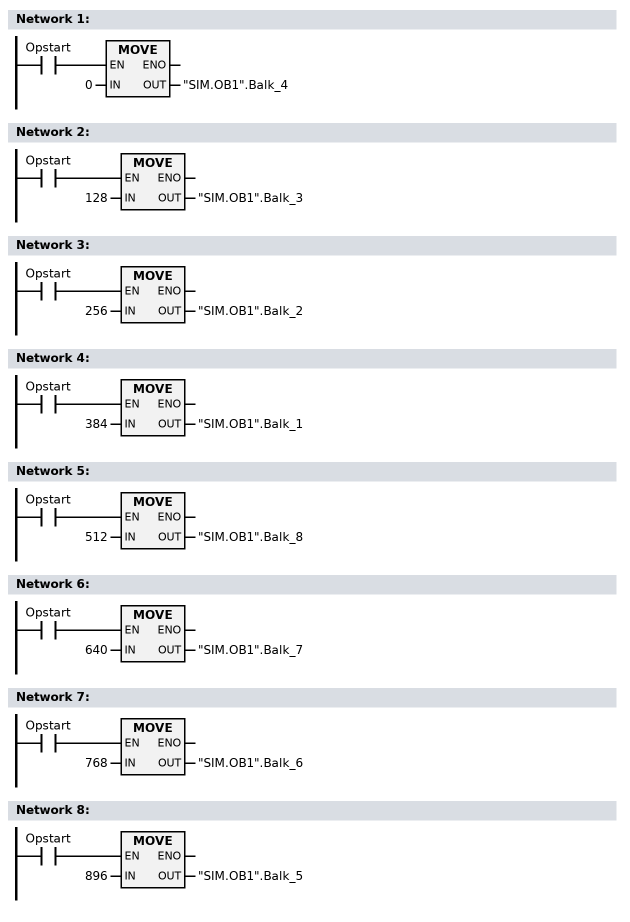
NETWORK
TITLE =
      A     "Opstart";
      JNB   _001;
      L     0;
      T     "SIM.OB1".Balk_4;
_001: NOP   0;
NETWORK
TITLE =
      A     "Opstart";
      JNB   _002;
      L     128;
      T     "SIM.OB1".Balk_3;
_002: NOP   0;
NETWORK
TITLE =
      A     "Opstart";
      JNB   _003;
      L     256;
      T     "SIM.OB1".Balk_2;
_003: NOP   0;
NETWORK
TITLE =
      A     "Opstart";
      JNB   _004;
      L     384;
      T     "SIM.OB1".Balk_1;
_004: NOP   0;
NETWORK
TITLE =
      A     "Opstart";
      JNB   _005;
      L     512;
      T     "SIM.OB1".Balk_8;
_005: NOP   0;
NETWORK
TITLE =
      A     "Opstart";
      JNB   _006;
      L     640;
      T     "SIM.OB1".Balk_7;
_006: NOP   0;
NETWORK
TITLE =
      A     "Opstart";
      JNB   _007;
      L     768;
      T     "SIM.OB1".Balk_6;
_007: NOP   0;
NETWORK
TITLE =
      A     "Opstart";
      JNB   _008;
      L     896;
      T     "SIM.OB1".Balk_5;
_008: NOP   0;
END_FUNCTION

FUNCTION "SIM.user" : VOID	// FC 11
VERSION : 0.1
BEGIN
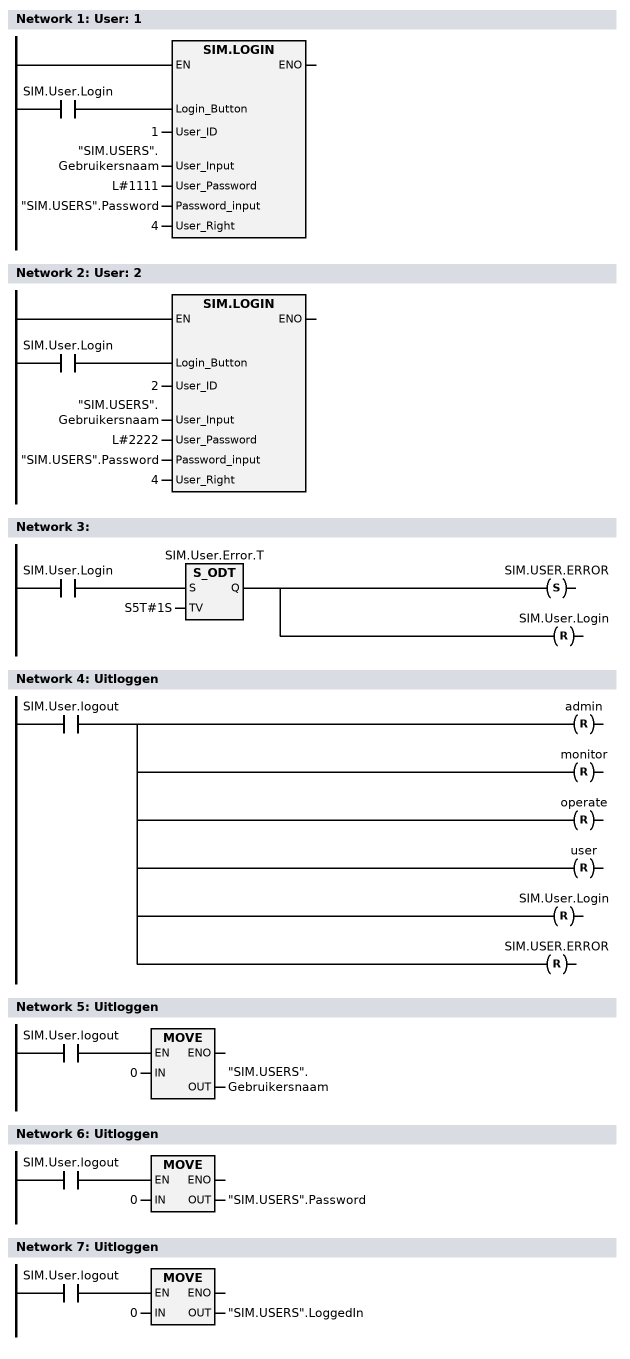
NETWORK
TITLE = User: 1
      A     "SIM.User.Login";
      =     L 0.0;
      BLD   103;
      CALL  "SIM.LOGIN" (
           Login_Button             := L 0.0,
           User_ID                  := 1,
           User_Input               := "SIM.USERS".Gebruikersnaam,
           User_Password            := L#1111,
           Password_input           := "SIM.USERS".Password,
           User_Right               := 4);
      NOP   0;
NETWORK
TITLE = User: 2
      A     "SIM.User.Login";
      =     L 0.0;
      BLD   103;
      CALL  "SIM.LOGIN" (
           Login_Button             := L 0.0,
           User_ID                  := 2,
           User_Input               := "SIM.USERS".Gebruikersnaam,
           User_Password            := L#2222,
           Password_input           := "SIM.USERS".Password,
           User_Right               := 4);
      NOP   0;
NETWORK
TITLE =
      A     "SIM.User.Login";
      L     S5T#1S;
      SD    "SIM.User.Error.T";
      NOP   0;
      NOP   0;
      NOP   0;
      A     "SIM.User.Error.T";
      S     "SIM.USER.ERROR";
      R     "SIM.User.Login";
NETWORK
TITLE = Uitloggen
      A     "SIM.User.logout";
      R     "admin";
      R     "monitor";
      R     "operate";
      R     "user";
      R     "SIM.User.Login";
      R     "SIM.USER.ERROR";
NETWORK
TITLE = Uitloggen
      A     "SIM.User.logout";
      JNB   _001;
      L     0;
      T     "SIM.USERS".Gebruikersnaam;
_001: NOP   0;
NETWORK
TITLE = Uitloggen
      A     "SIM.User.logout";
      JNB   _002;
      L     0;
      T     "SIM.USERS".Password;
_002: NOP   0;
NETWORK
TITLE = Uitloggen
      A     "SIM.User.logout";
      JNB   _003;
      L     0;
      T     "SIM.USERS".LoggedIn;
_003: NOP   0;
END_FUNCTION

FUNCTION "Positionering_balken" : VOID	// FC 12
VERSION : 0.1
BEGIN
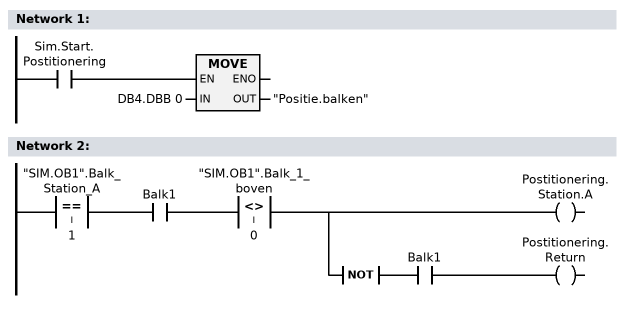
NETWORK
TITLE =
      A     "Sim.Start.Postitionering";
      JNB   _001;
      L     DB4.DBB 0;
      T     "Positie.balken";
_001: NOP   0;
NETWORK
TITLE =
      A(;
      L     "SIM.OB1".Balk_Station_A;
      L     1;
      ==I;
      );
      A     "Balk1";
      A(;
      L     "SIM.OB1".Balk_1_boven;
      L     0;
      <>I;
      );
      =     L 0.0;
      A     L 0.0;
      BLD   102;
      =     "Postitionering.Station.A";
      A     L 0.0;
      NOT;
      A     "Balk1";
      =     "Postitionering.Return";
END_FUNCTION

FUNCTION "Sub_routine" : VOID	// FC 14
VERSION : 0.1
VAR_INPUT
  voorwaarde : BOOL ;
END_VAR
VAR_IN_OUT
  huidige : BOOL ;
  volgende : BOOL ;
END_VAR
BEGIN
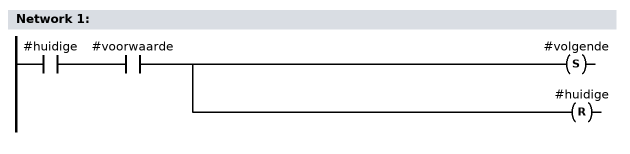
NETWORK
TITLE =
      A     #huidige;
      A     #voorwaarde;
      S     #volgende;
      R     #huidige;
END_FUNCTION

FUNCTION "Opstart_subroutine" : VOID	// FC 15
VERSION : 0.1
VAR_INPUT
  voorwaarde : BOOL ;
END_VAR
VAR_IN_OUT
  huidige : BOOL ;
  volgende_1 : BOOL ;
  volgende_2 : BOOL ;
END_VAR
BEGIN
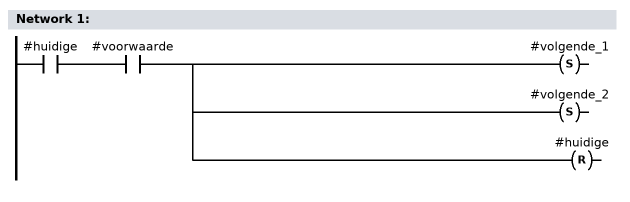
NETWORK
TITLE =
      A     #huidige;
      A     #voorwaarde;
      S     #volgende_1;
      S     #volgende_2;
      R     #huidige;
END_FUNCTION

FUNCTION "Sub_routine_gelijk" : VOID	// FC 16
VERSION : 0.1
VAR_INPUT
  voorwaarde : BOOL ;
END_VAR
VAR_IN_OUT
  huidige : BOOL ;
  volgende_1 : BOOL ;
  volgende_2 : BOOL ;
END_VAR
BEGIN
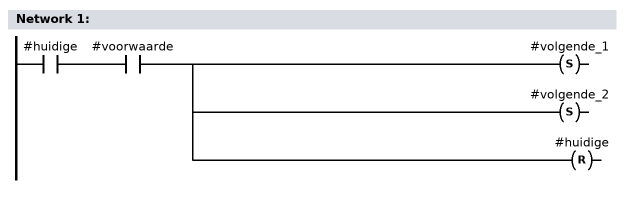
NETWORK
TITLE =
      A     #huidige;
      A     #voorwaarde;
      S     #volgende_1;
      S     #volgende_2;
      R     #huidige;
END_FUNCTION

FUNCTION "Sub_route_Station_samen" : VOID	// FC 17
VERSION : 0.1
VAR_INPUT
  voorwaarde : BOOL ;
END_VAR
VAR_IN_OUT
  huidige : BOOL ;
  volgende_1 : BOOL ;
  volgende_2 : BOOL ;
  volgende_3 : BOOL ;
END_VAR
BEGIN
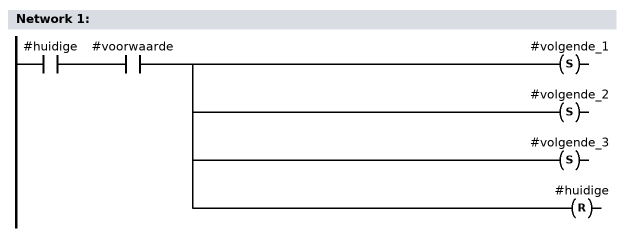
NETWORK
TITLE =
      A     #huidige;
      A     #voorwaarde;
      S     #volgende_1;
      S     #volgende_2;
      S     #volgende_3;
      R     #huidige;
END_FUNCTION

FUNCTION FC 18 : VOID
VERSION : 0.1
VAR_INPUT
  voorwaarde : BOOL ;
END_VAR
VAR_IN_OUT
  huidige_1 : BOOL ;
  huidige_2 : BOOL ;
  volgende : BOOL ;
END_VAR
BEGIN
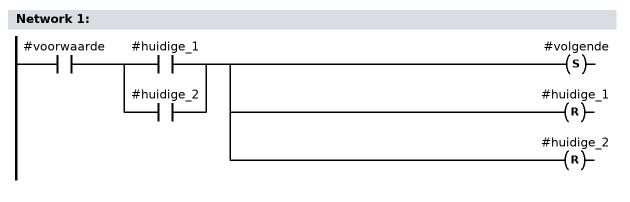
NETWORK
TITLE =
      A     #voorwaarde;
      A(;
      O     #huidige_1;
      O     #huidige_2;
      );
      S     #volgende;
      R     #huidige_1;
      R     #huidige_2;
END_FUNCTION

FUNCTION "SIM.SUBR.Y-As" : VOID	// FC 19
VERSION : 0.1
VAR_INPUT
  Balk_nr : INT ;
END_VAR
VAR_IN_OUT
  DB_Balk : INT ;
END_VAR
VAR_TEMP
  Timer2 : BOOL ;
  Timer1 : BOOL ;
  StationA : BOOL ;
  StationB : BOOL ;
END_VAR
BEGIN
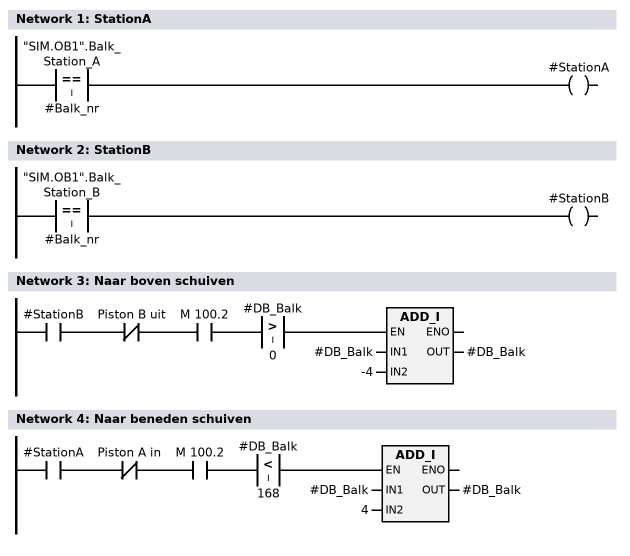
NETWORK
TITLE = StationA
      L     "SIM.OB1".Balk_Station_A;
      L     #Balk_nr;
      ==I;
      =     #StationA;
NETWORK
TITLE = StationB
      L     "SIM.OB1".Balk_Station_B;
      L     #Balk_nr;
      ==I;
      =     #StationB;
NETWORK
TITLE = Naar boven schuiven
      A     #StationB;
      AN    "Piston B uit";
      A     M 100.2;
      A(;
      L     #DB_Balk;
      L     0;
      >I;
      );
      JNB   _001;
      L     #DB_Balk;
      L     -4;
      +I;
      T     #DB_Balk;
_001: NOP   0;
NETWORK
TITLE = Naar beneden schuiven
      A     #StationA;
      AN    "Piston A in";
      A     M 100.2;
      A(;
      L     #DB_Balk;
      L     168;
      <I;
      );
      JNB   _002;
      L     #DB_Balk;
      L     4;
      +I;
      T     #DB_Balk;
_002: NOP   0;
END_FUNCTION

FUNCTION "SIM.LOGIN" : VOID	// FC 20
VERSION : 0.1
VAR_INPUT
  Login_Button : BOOL ;
  User_ID : INT ;
  User_Input : INT ;
  User_Password : DINT ;
  Password_input : DINT ;
  User_Right : INT ;
END_VAR
VAR_TEMP
  ID_OF_Input : BOOL ;
  Password_Correct : BOOL ;
END_VAR
BEGIN
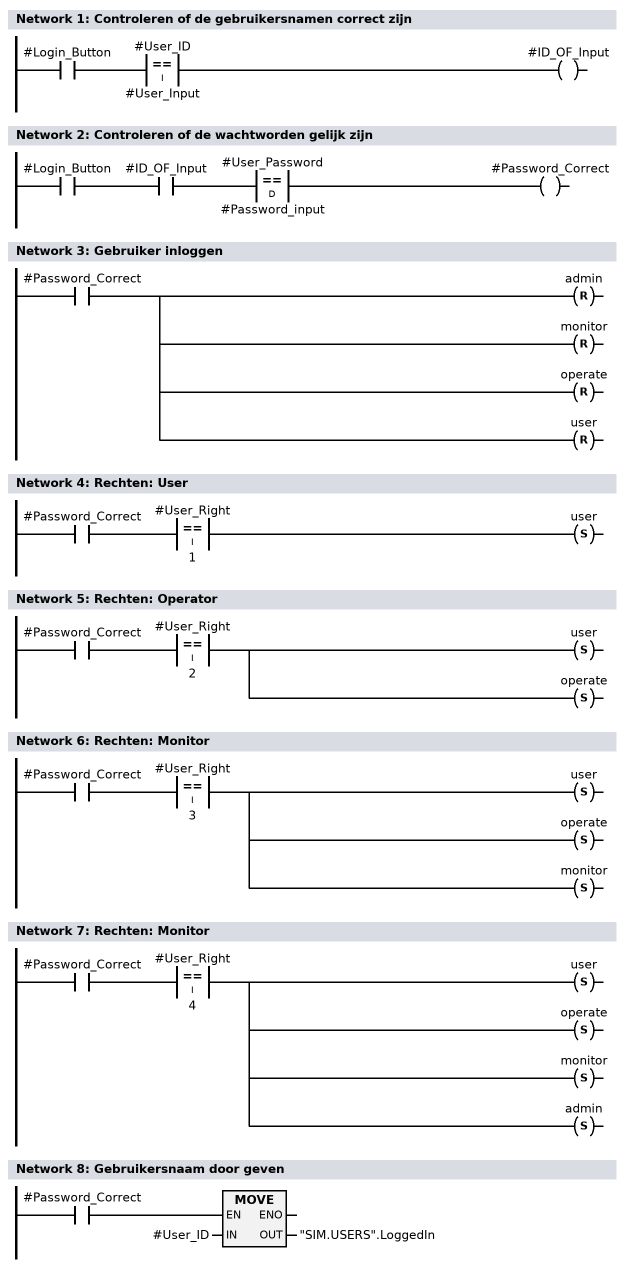
NETWORK
TITLE = Controleren of de gebruikersnamen correct zijn
      A     #Login_Button;
      A(;
      L     #User_ID;
      L     #User_Input;
      ==I;
      );
      =     #ID_OF_Input;
NETWORK
TITLE = Controleren of de wachtworden gelijk zijn
      A     #Login_Button;
      A     #ID_OF_Input;
      A(;
      L     #User_Password;
      L     #Password_input;
      ==D;
      );
      =     #Password_Correct;
NETWORK
TITLE = Gebruiker inloggen
      A     #Password_Correct;
      R     "admin";
      R     "monitor";
      R     "operate";
      R     "user";
NETWORK
TITLE = Rechten: User
      A     #Password_Correct;
      A(;
      L     #User_Right;
      L     1;
      ==I;
      );
      S     "user";
NETWORK
TITLE = Rechten: Operator
      A     #Password_Correct;
      A(;
      L     #User_Right;
      L     2;
      ==I;
      );
      S     "user";
      S     "operate";
NETWORK
TITLE = Rechten: Monitor
      A     #Password_Correct;
      A(;
      L     #User_Right;
      L     3;
      ==I;
      );
      S     "user";
      S     "operate";
      S     "monitor";
NETWORK
TITLE = Rechten: Monitor
      A     #Password_Correct;
      A(;
      L     #User_Right;
      L     4;
      ==I;
      );
      S     "user";
      S     "operate";
      S     "monitor";
      S     "admin";
NETWORK
TITLE = Gebruikersnaam door geven
      A     #Password_Correct;
      JNB   _001;
      L     #User_ID;
      T     "SIM.USERS".LoggedIn;
_001: NOP   0;
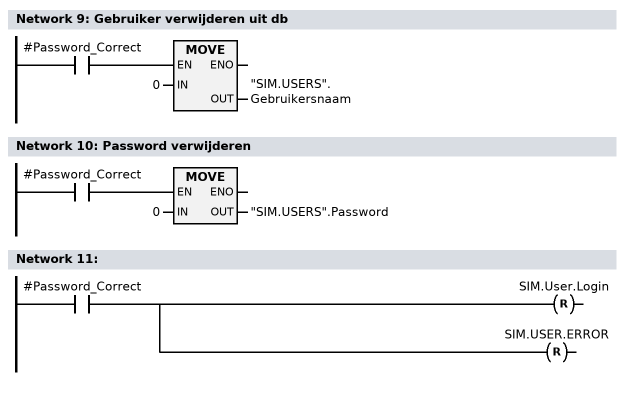
NETWORK
TITLE = Gebruiker verwijderen uit db
      A     #Password_Correct;
      JNB   _002;
      L     0;
      T     "SIM.USERS".Gebruikersnaam;
_002: NOP   0;
NETWORK
TITLE = Password verwijderen
      A     #Password_Correct;
      JNB   _003;
      L     0;
      T     "SIM.USERS".Password;
_003: NOP   0;
NETWORK
TITLE =
      A     #Password_Correct;
      R     "SIM.User.Login";
      R     "SIM.USER.ERROR";
END_FUNCTION

FUNCTION "SIM.Move.X-As" : VOID	// FC 21
VERSION : 0.1
VAR_INPUT
  Sensor : BOOL ;
  Xvalue : INT ;
END_VAR
BEGIN
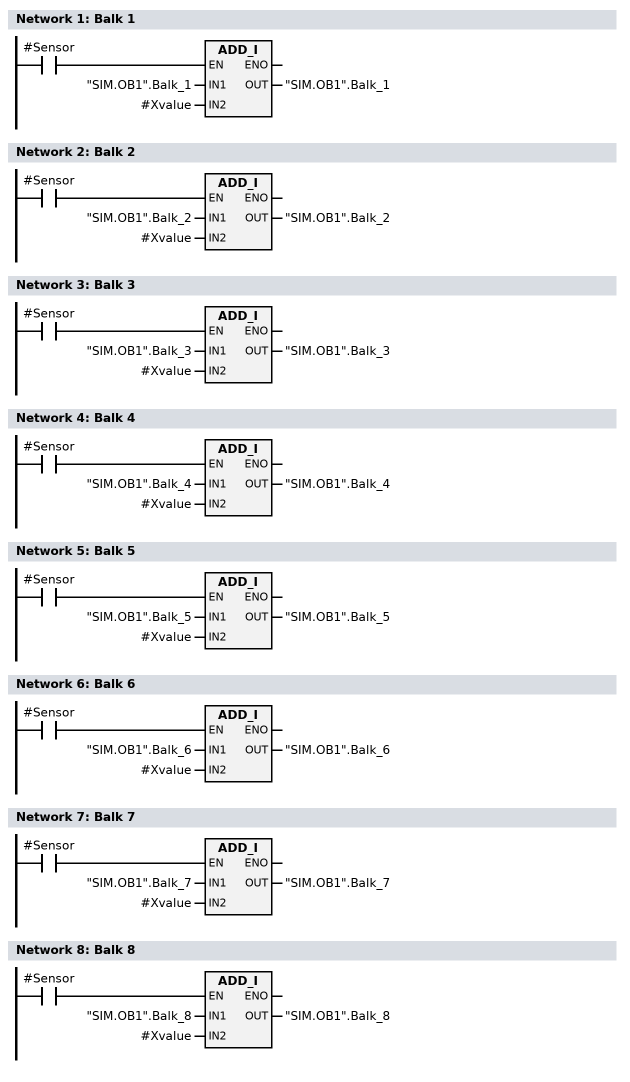
NETWORK
TITLE = Balk 1
      A     #Sensor;
      JNB   _001;
      L     "SIM.OB1".Balk_1;
      L     #Xvalue;
      +I;
      T     "SIM.OB1".Balk_1;
_001: NOP   0;
NETWORK
TITLE = Balk 2
      A     #Sensor;
      JNB   _002;
      L     "SIM.OB1".Balk_2;
      L     #Xvalue;
      +I;
      T     "SIM.OB1".Balk_2;
_002: NOP   0;
NETWORK
TITLE = Balk 3
      A     #Sensor;
      JNB   _003;
      L     "SIM.OB1".Balk_3;
      L     #Xvalue;
      +I;
      T     "SIM.OB1".Balk_3;
_003: NOP   0;
NETWORK
TITLE = Balk 4
      A     #Sensor;
      JNB   _004;
      L     "SIM.OB1".Balk_4;
      L     #Xvalue;
      +I;
      T     "SIM.OB1".Balk_4;
_004: NOP   0;
NETWORK
TITLE = Balk 5
      A     #Sensor;
      JNB   _005;
      L     "SIM.OB1".Balk_5;
      L     #Xvalue;
      +I;
      T     "SIM.OB1".Balk_5;
_005: NOP   0;
NETWORK
TITLE = Balk 6
      A     #Sensor;
      JNB   _006;
      L     "SIM.OB1".Balk_6;
      L     #Xvalue;
      +I;
      T     "SIM.OB1".Balk_6;
_006: NOP   0;
NETWORK
TITLE = Balk 7
      A     #Sensor;
      JNB   _007;
      L     "SIM.OB1".Balk_7;
      L     #Xvalue;
      +I;
      T     "SIM.OB1".Balk_7;
_007: NOP   0;
NETWORK
TITLE = Balk 8
      A     #Sensor;
      JNB   _008;
      L     "SIM.OB1".Balk_8;
      L     #Xvalue;
      +I;
      T     "SIM.OB1".Balk_8;
_008: NOP   0;
END_FUNCTION

FUNCTION "SIM.BALK.Reset" : VOID	// FC 22
VERSION : 0.1
VAR_IN_OUT
  Balk : INT ;
END_VAR
BEGIN
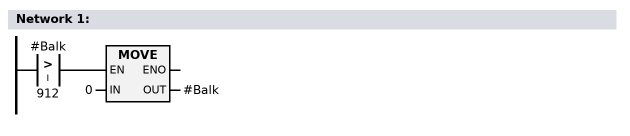
NETWORK
TITLE =
      A(;
      L     #Balk;
      L     912;
      >I;
      );
      JNB   _001;
      L     0;
      T     #Balk;
_001: NOP   0;
END_FUNCTION

DATA_BLOCK DB 1
VERSION : 0.1
  STRUCT
   Ingevoerde_Waarde : INT ;
   Momentele_Waarde : INT ;
  END_STRUCT ;	
BEGIN
END_DATA_BLOCK

DATA_BLOCK "SIM.OB1"	// DB 2
VERSION : 0.1
  STRUCT
   Balk_1 : INT ;	//0
   Balk_2 : INT ;	//0
   Balk_3 : INT ;	//0
   Balk_4 : INT ;	//0
   Balk_5 : INT ;	//0
   Balk_6 : INT ;	//0
   Balk_7 : INT ;	//0
   Balk_8 : INT ;	//0
   Balk_1_boven : INT ;	//0
   Balk_2_boven : INT ;
   Balk_3_boven : INT ;
   Balk_4_boven : INT ;
   Balk_5_boven : INT ;
   Balk_6_boven : INT ;
   Balk_7_boven : INT ;
   Balk_8_boven : INT ;
   Balk_Sensoren : INT ;
   Balk_Station_A : INT ;
   Balk_Station_B : INT ;
   Balk_Station_A_Mom : INT ;	//Momentele waarde
   Balk_Station_B_Mom : INT ;	//Momentele waarde
  END_STRUCT ;	
BEGIN
END_DATA_BLOCK

DATA_BLOCK "SIM.USERS"	// DB 3
VERSION : 0.1
  STRUCT
   Gebruikersnaam : INT ;	//Temporary placeholder variable
   Password : DINT ;
   LoggedIn : INT ;
  END_STRUCT ;	
BEGIN
END_DATA_BLOCK

DATA_BLOCK "Positionering"	// DB 4
VERSION : 0.1
  STRUCT
   Balk_1 : BOOL ;	//Temporary placeholder variable
   Balk_2 : BOOL ;
   Balk_3 : BOOL ;
   Balk_4 : BOOL ;
   Balk_5 : BOOL ;
   Balk_6 : BOOL ;
   Balk_7 : BOOL ;
   Balk_8 : BOOL ;
   Recept1 : BYTE ;
   Recept2 : BYTE ;
   Recept3 : BYTE ;
   Recept4 : BYTE ;
   Recept5 : BYTE ;
   Recept6 : BYTE ;
   Recept7 : BYTE ;
   Recept8 : BYTE ;
   Recept9 : BYTE ;
   Recept10 : BYTE ;
   Recept_Save : INT ;
   Recept_Zoom : INT ;
  END_STRUCT ;	
BEGIN
END_DATA_BLOCK

ORGANIZATION_BLOCK OB 1
TITLE = "Main Program Sweep (Cycle)"
VERSION : 0.1
VAR_TEMP
  OB1_EV_CLASS : BYTE ;	//Bits 0-3 = 1 (Coming event), Bits 4-7 = 1 (Event class 1)
  OB1_SCAN_1 : BYTE ;	//1 (Cold restart scan 1 of OB 1), 3 (Scan 2-n of OB 1)
  OB1_PRIORITY : BYTE ;	//Priority of OB Execution
  OB1_OB_NUMBR : BYTE ;	//1 (Organization block 1, OB1)
  OB1_RESERVED_1 : BYTE ;	//Reserved for system
  OB1_RESERVED_2 : BYTE ;	//Reserved for system
  OB1_PREV_CYCLE : INT ;	//Cycle time of previous OB1 scan (milliseconds)
  OB1_MIN_CYCLE : INT ;	//Minimum cycle time of OB1 (milliseconds)
  OB1_MAX_CYCLE : INT ;	//Maximum cycle time of OB1 (milliseconds)
  OB1_DATE_TIME : DATE_AND_TIME ;	//Date and time OB1 started
END_VAR
BEGIN
NETWORK
TITLE =
      CALL  "Uitgangen Sturen";
      CALL  "DB_Function";
      CALL  "Timers + Counters";
      CALL  "Simulatie_Run";
      CALL  "Opstart_FC";
      CALL  "SIM.OB100";
      CALL  "SIM.user";
      CALL  "Positionering_balken";
      CALL  "Grafcet_Platform";
      CALL  "Grafcet Station A";
      CALL  "Grafcet Station B";
      CALL  "Ingang -> Merker";
END_ORGANIZATION_BLOCK

ORGANIZATION_BLOCK "COMPLETE RESTART"	// OB 100
TITLE = "Complete Restart"
VERSION : 0.1
VAR_TEMP
  OB100_EV_CLASS : BYTE ;	//16#13, Event class 1, Entering event state, Event logged in diagnostic buffer
  OB100_STRTUP : BYTE ;	//16#81/82/83/84 Method of startup
  OB100_PRIORITY : BYTE ;	//Priority of OB Execution
  OB100_OB_NUMBR : BYTE ;	//100 (Organization block 100, OB100)
  OB100_RESERVED_1 : BYTE ;	//Reserved for system
  OB100_RESERVED_2 : BYTE ;	//Reserved for system
  OB100_STOP : WORD ;	//Event that caused CPU to stop (16#4xxx)
  OB100_STRT_INFO : DWORD ;	//Information on how system started
  OB100_DATE_TIME : DATE_AND_TIME ;	//Date and time OB100 started
END_VAR
BEGIN
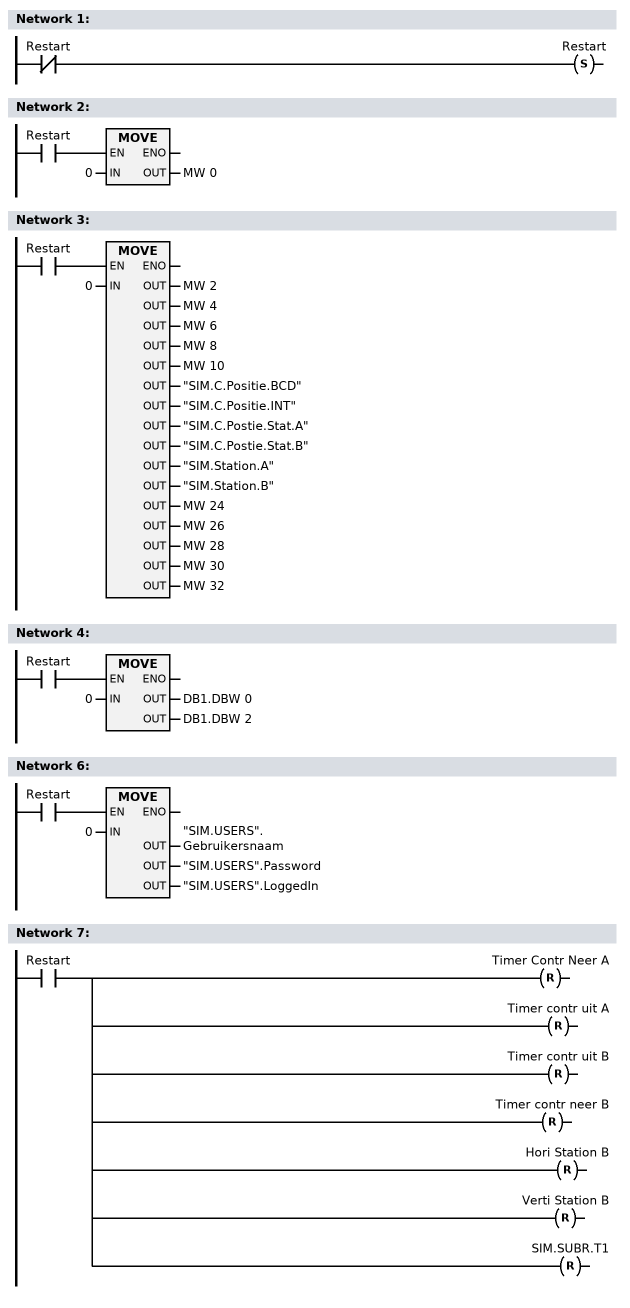
NETWORK
TITLE =
      AN    "Restart";
      S     "Restart";
NETWORK
TITLE =
      A     "Restart";
      JNB   _001;
      L     0;
      T     MW 0;
_001: NOP   0;
NETWORK
TITLE =
      A     "Restart";
      JNB   _002;
      L     0;
      T     MW 2;
      T     MW 4;
      T     MW 6;
      T     MW 8;
      T     MW 10;
      T     "SIM.C.Positie.BCD";
      T     "SIM.C.Positie.INT";
      T     "SIM.C.Postie.Stat.A";
      T     "SIM.C.Postie.Stat.B";
      T     "SIM.Station.A";
      T     "SIM.Station.B";
      T     MW 24;
      T     MW 26;
      T     MW 28;
      T     MW 30;
      T     MW 32;
_002: NOP   0;
NETWORK
TITLE =
      A     "Restart";
      JNB   _003;
      L     0;
      T     DB1.DBW 0;
      T     DB1.DBW 2;
_003: NOP   0;
NETWORK
TITLE =
      A     "Restart";
      JNB   _003;
      L     0;
      T     "SIM.OB1".Balk_1;
      T     "SIM.OB1".Balk_2;
      T     "SIM.OB1".Balk_3;
      T     "SIM.OB1".Balk_4;
      T     "SIM.OB1".Balk_5;
      T     "SIM.OB1".Balk_6;
      T     "SIM.OB1".Balk_7;
      T     "SIM.OB1".Balk_8;
      T     "SIM.OB1".Balk_1_boven;
      T     "SIM.OB1".Balk_2_boven;
      T     "SIM.OB1".Balk_3_boven;
      T     "SIM.OB1".Balk_4_boven;
      T     "SIM.OB1".Balk_5_boven;
      T     "SIM.OB1".Balk_6_boven;
      T     "SIM.OB1".Balk_7_boven;
      T     "SIM.OB1".Balk_8_boven;
NETWORK
TITLE =
      A     "Restart";
      JNB   _004;
      L     0;
      T     "SIM.USERS".Gebruikersnaam;
      T     "SIM.USERS".Password;
      T     "SIM.USERS".LoggedIn;
_004: NOP   0;
NETWORK
TITLE =
      A     "Restart";
      R     "Timer Contr Neer A";
      R     "Timer contr uit A";
      R     "Timer contr uit B";
      R     "Timer contr neer B";
      R     "Hori Station B";
      R     "Verti Station B";
      R     "SIM.SUBR.T1";
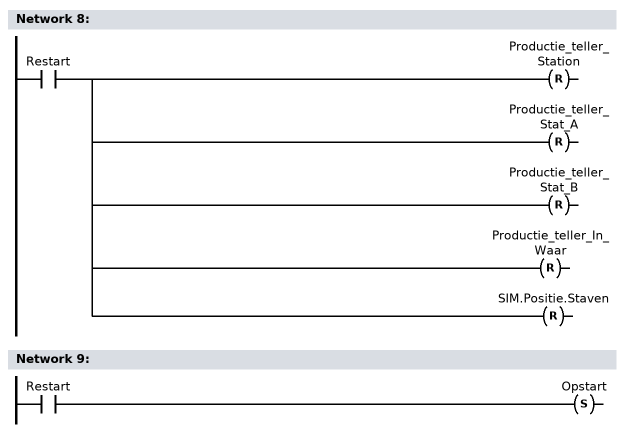
NETWORK
TITLE =
      A     "Restart";
      R     "Productie_teller_Station";
      R     "Productie_teller_Stat_A";
      R     "Productie_teller_Stat_B";
      R     "Productie_teller_In_Waar";
      R     "SIM.Positie.Staven";
NETWORK
TITLE =
      A     "Restart";
      S     "Opstart";
END_ORGANIZATION_BLOCK

SYMBOL_TABLE
"Counter.Balk"	C 0	COUNTER
"Geheugen.Platform"	DB 1	DB 1
"Geheugen.Instellingen"	DB 2	DB 2
"Uitgangen.Sturen"	FC 1	FC 1
"Merkers.Sturen"	FC 2	FC 2
"Timers + Counters"	FC 3	FC 3
"Berekeningen"	FC 4	FC 4
"Grafcet"	FC 5	FC 5
"Simulatie"	FC 6	FC 6
"Watch.Dog"	FC 7	FC 7
"Sub.Basis"	FC 14	FC 14
"Sub.Keuze"	FC 15	FC 15
"Sub.Keuze.Sta.A.or.B"	FC 16	FC 16
"Stap 0.0"	M 0.0	BOOL
"Stap 0.1"	M 0.1	BOOL
"Stap 0.2"	M 0.2	BOOL
"Stap 0.3"	M 0.3	BOOL
"Stap 0.4"	M 0.4	BOOL
"Stap 0.5"	M 0.5	BOOL
"Stap 0.6"	M 0.6	BOOL
"Stap 0.7"	M 0.7	BOOL
"Stap 1.0"	M 1.0	BOOL
"Stap 1.1"	M 1.1	BOOL
"Stap 1.2"	M 1.2	BOOL
"Stap 1.3"	M 1.3	BOOL
"Stap 1.4"	M 1.4	BOOL
"Stap 1.5"	M 1.5	BOOL
"Stap 1.6"	M 1.6	BOOL
"Stap 1.7"	M 1.7	BOOL
"Stap 2.0"	M 2.0	BOOL
"Stap 2.1"	M 2.1	BOOL
"Stap 2.2"	M 2.2	BOOL
"Stap 2.3"	M 2.3	BOOL
"Stap 2.4"	M 2.4	BOOL
"Stap 2.5"	M 2.5	BOOL
"Stap 2.6"	M 2.6	BOOL
"Stap 2.7"	M 2.7	BOOL
"Stap 3.0"	M 3.0	BOOL
"Stap 3.1"	M 3.1	BOOL
"Stap 3.2"	M 3.2	BOOL
"Stap 3.3"	M 3.3	BOOL
"Stap 3.4"	M 3.4	BOOL
"Stap 3.5"	M 3.5	BOOL
"Stap 3.6"	M 3.6	BOOL
"Stap 3.7"	M 3.7	BOOL
"Stap 4.0"	M 4.0	BOOL
"Stap 4.1"	M 4.1	BOOL
"Stap 4.2"	M 4.2	BOOL
"Stap 4.3"	M 4.3	BOOL
"Stap 4.4"	M 4.4	BOOL
"Stap 4.5"	M 4.5	BOOL
"Stap 4.6"	M 4.6	BOOL
"Stap 4.7"	M 4.7	BOOL
"Stop.Hardware"	M 10.0	BOOL
"Start.Hardware"	M 10.1	BOOL
"Sens.Sta.A.In"	M 10.2	BOOL
"Sens.Sta.A.Forward"	M 10.3	BOOL
"Sens.Sta.A.Down"	M 10.4	BOOL
"Sens.Sta.A.Up"	M 10.5	BOOL
"Sens.Sta.B.In"	M 10.6	BOOL
"Sens.Sta.B.Forward"	M 10.7	BOOL
"Sens.Sta.B.Down"	M 11.0	BOOL
"Sens.Sta.B.Up"	M 11.1	BOOL
"Sens.Proxi.1"	M 11.2	BOOL
"Sens.Proxi.2"	M 11.3	BOOL
"NoodStop.Relais"	M 11.4	BOOL
"Leeg"	M 12.0	BOOL
"Motor.Platform.Rechts"	M 12.1	BOOL
"Station.A.Down"	M 12.2	BOOL
"Station.A.Forward"	M 12.3	BOOL
"Station.B.Down"	M 12.4	BOOL
"Station.B.In"	M 12.5	BOOL
"Sign.Rood"	M 12.6	BOOL
"Sign.Groen"	M 12.7	BOOL
"Motor.Platform.Links"	M 13.0	BOOL
"Opstart.Cycle"	M 14.0	BOOL
"Sim.start"	M 14.1	BOOL
"Sim.Reset"	M 14.2	BOOL
"Restart"	M 14.3	BOOL
"Stop.Cycle"	M 14.4	BOOL
"Restart.Cycle"	M 14.5	BOOL
"Blinker.4s"	M 100.4	BOOL
"Blinker.5s"	M 100.5	BOOL
"Blinker.6s"	M 100.6	BOOL
"Restart.OB100"	M 101.0	BOOL
"Ingangen I0.x"	MB 10	BYTE
"Ingangen I124.x"	MB 11	BYTE
"Uitgangen Q0.x"	MB 12	BYTE
"Uitgangen Q124.x"	MB 13	BYTE
"Blinkers"	MB 100	BYTE
"Programma.Cyclus"	OB 1	OB 1
"COMPLETE RESTART"	OB 100	OB 100	// Complete Restart
"Motor.Check"	T 0	TIMER
"Platform.Vertraging"	T 1	TIMER
END_SYMBOL_TABLE

SYMBOL_TABLE
"I/O.Send"	FC 1	FC 1
"Noodstop.relais"	I 124.4	BOOL
"IB0"	MB 10	BYTE
"IB124"	MB 11	BYTE
"QB0"	MB 12	BYTE
"QB124"	MB 13	BYTE
"Programma.Cyclus"	OB 1	OB 1
END_SYMBOL_TABLE
